// TwinCAT 3 PLC project PlcTc3JsonXmlSampleJsonSaxWriter
// ProgramVersion: 3.1.4021.2
// libraries:
//   Tc2_Standard, * (Beckhoff Automation GmbH)
//   Tc2_System, * (Beckhoff Automation GmbH)
//   Tc3_JsonXml, * (Beckhoff Automation GmbH)
//   Tc3_Module, * (Beckhoff Automation GmbH)
// project tree:
//   / PlcTask.TcTTO
//   POUs/ MAIN.TcPOU
// real-time tasks:
//   TASK PlcTask: cycle T#10ms, priority 20, ADS port 350

CONFIGURATION PlcTc3JsonXmlSampleJsonSaxWriter
    RESOURCE PLC ON TwinCAT3
        TASK PlcTask(INTERVAL := T#10ms, PRIORITY := 20);
        PROGRAM MAIN WITH PlcTask : MAIN;
    END_RESOURCE
END_CONFIGURATION

// ---- POUs/MAIN.TcPOU
PROGRAM MAIN
VAR
	dtTimestamp : DATE_AND_TIME := DT#2017-04-04-12:42:42;
  	(* JSON document *)
	fbJson 		: FB_JsonSaxWriter;
	sJsonDoc 	: STRING(255);
END_VAR

fbJson.StartObject();
fbJson.AddKey('Values');
fbJson.StartObject();
fbJson.AddKey('Timestamp');
fbJson.AddDateTime(dtTimestamp);
fbJson.AddKey('Sensor1');
fbJson.AddReal(42.42);
fbJson.AddKey('Sensor2');
fbJson.AddDint(42);
fbJson.AddKey('Sensor3');
fbJson.AddBool(TRUE);
fbJson.EndObject();
fbJson.EndObject();
sJsonDoc := fbJson.GetDocument();
fbJson.ResetDocument();

END_PROGRAM
